FUNCTION_BLOCK FB_Dictionary IMPLEMENTS I_Dictionary
VAR_INPUT
END_VAR
VAR_OUTPUT
END_VAR
VAR
	bAdd:				BOOL;
	bReset:				Bool;
	bLoad:				BOOL;
	bSave:				BOOL;
	fbJson:				FB_JsonDomParser;
  	jObject:				SJsonValue;
	
	sJson: 				STRING(255);
END_VAR

IF bReset THEN
	bReset:= FALSE;
	jObject:= fbJson.NewDocument();
	bSave:= TRUE;
END_IF

IF bAdd THEN
	// How to parse instace path?
	M_Add('member.Value1', 'Value1');
	M_Add('member.Value2', 'Value2');
	
END_IF

//jMember:= fbJson.FindMemberPath(jObject,'/member/Value1');



fbJson.LoadDocumentFromFile('C:\Test.json', bLoad);

fbJson.SaveDocumentToFile('C:\Test.json', bSave);


fbJson.CopyDocument(sJson, SIZEOF(sJson));

METHOD PUBLIC M_Add : BOOL
VAR_INPUT
	Key:		STRING(255);
	Value:		STRING(255);
END_VAR
VAR 
	sKey:			STRING(255);
	sMember:		STRING(255);
  	jMember:		SJsonValue;
	nPosition:		INT;
END_VAR
sKey:= Key;
nPosition:= FIND(sKey, '.');
WHILE ( nPosition <> 0) DO
	sMember:= LEFT(sKey, nPosition - 1);
	IF fbJson.HasMember(jObject, Key) THEN
		;
	ELSE
		fbJson.AddStringMember(jObject, sMember, '');			
	END_IF

	sKey:= DELETE(sKey, nPosition, 1);
	nPosition:= FIND(sKey, '.');
	IF nPosition = 0 THEN
		fbJson.AddStringMember(jObject, sKey, Value);	
	END_IF
END_WHILE


//IF fbJson.HasMember(jObject, Key) = 0 THEN
//	fbJson.AddStringMember(jObject, Key, Value);		
//END_IF
END_METHOD

METHOD PUBLIC M_GetSTRING : String(255)
VAR_INPUT
	sName:	STRING(255);
END_VAR
END_METHOD

METHOD PUBLIC M_Load : BOOL
VAR_INPUT
	sFile:	STRING(255);
END_VAR
END_METHOD

METHOD PUBLIC M_Reset : BOOL
VAR_INPUT
END_VAR
END_METHOD

METHOD PUBLIC M_Save : BOOL
VAR_INPUT
END_VAR
END_METHOD

END_FUNCTION_BLOCK

(* stored: Version 1.1.0.1
   POU FB_Dictionary: Id {ca35913f-5cdc-0fb1-22b9-4c30741035cf}, SpecialFunc None
   Method M_Add: Id {5f198432-6b9a-0cc9-223e-32fac07c9c15}
   Method M_GetSTRING: Id {36d7e4d9-6385-0d15-1db3-61b9b3f66c18}
   Method M_Load: Id {0cfe07f9-80a6-0092-1199-05d47a634bea}
   Method M_Reset: Id {a41c1e35-f20d-09aa-09c0-ce2dae9cb17d}
   Method M_Save: Id {f15ba428-e316-0337-1810-7cf2e63511bb} *)
